FUNCTION_BLOCK AccumDDHHMM
VAR_INPUT
	State: BOOL;
	Retentive: BOOL;
	Reset:BOOL;
END_VAR

VAR PERSISTENT
	Mins: WORD;
	Hrs:  WORD;
	Days: WORD;	
END_VAR
VAR
	DisplayTime: STRING;
	timer: TON;
	timerPT: TIME:= T#1M;
	StateToOff: F_TRIG;
END_VAR

VAR_TEMP
	displayTimeFormat: FB_FormatString;
END_VAR
VAR // added by the converter: edge detectors and wires of the graphical bodies
    _w1, _w2, _w3, _w4 : BOOL;
END_VAR

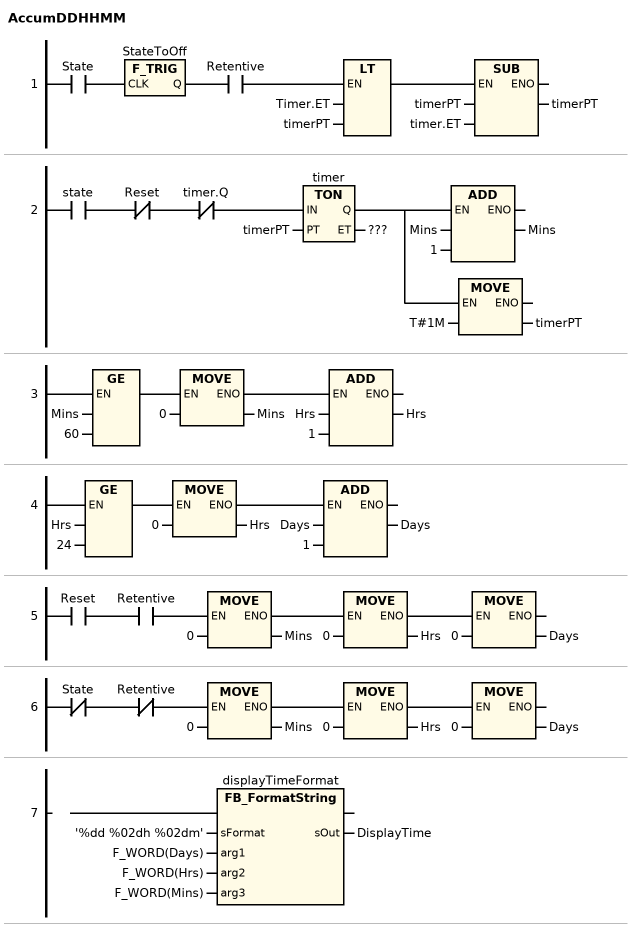
// NETWORK 1
StateToOff(CLK := State); // F_TRIG
IF StateToOff.Q AND Retentive AND Timer.ET < timerPT THEN timerPT := timerPT - timer.ET; END_IF

// NETWORK 2
timer(IN := state AND NOT Reset AND NOT timer.Q, PT := timerPT); // TON
IF timer.Q THEN Mins := Mins + 1; END_IF
IF timer.Q THEN timerPT := T#1M; END_IF

// NETWORK 3
_w1 := Mins >= 60;
IF _w1 THEN Mins := 0; END_IF
IF _w1 THEN Hrs := Hrs + 1; END_IF

// NETWORK 4
_w2 := Hrs >= 24;
IF _w2 THEN Hrs := 0; END_IF
IF _w2 THEN Days := Days + 1; END_IF

// NETWORK 5
_w3 := Reset AND Retentive;
IF _w3 THEN Mins := 0; END_IF
IF _w3 THEN Hrs := 0; END_IF
IF _w3 THEN Days := 0; END_IF

// NETWORK 6
_w4 := NOT State AND NOT Retentive;
IF _w4 THEN Mins := 0; END_IF
IF _w4 THEN Hrs := 0; END_IF
IF _w4 THEN Days := 0; END_IF

// NETWORK 7
displayTimeFormat(
    sFormat := '%dd %02dh %02dm',
    arg1 := F_WORD(Days),
    arg2 := F_WORD(Hrs),
    arg3 := F_WORD(Mins),
    sOut => DisplayTime); // FB_FormatString

END_FUNCTION_BLOCK

(* stored: Version 1.1.0.1, ProductVersion 3.1.4024.12
   POU AccumDDHHMM: Id {5199796b-956b-43e3-8121-00b9dc5b3dd7}, SpecialFunc None *)
